// Mitsubishi GX Works2 project: Embotido   PLC: FX1S

// global labels: Global1
VAR_GLOBAL
  Sensor1 AT X002 : BOOL;
  Sensor2 AT X003 : BOOL;
  Sensor3 AT X005 : BOOL;
  Sensor4 AT X004 : BOOL;
  btnStart AT X000 : BOOL;
  btnStop AT X001 : BOOL;
  btnManConveyor AT X012 : BOOL;
  btnManSolenoid2 AT X007 : BOOL;
  btnManSolenoid1 AT X006 : BOOL;
  btnManSolenoid3 AT X010 : BOOL;
  btnManSolenoid4 AT X011 : BOOL;
  LightSensor1O AT Y007 : BOOL;
  LightSensor2O AT Y010 : BOOL;
  LightSensor3O AT Y011 : BOOL;
  LightSensor4O AT Y012 : BOOL;
  LightStartO AT Y005 : BOOL;
  LightStopO AT Y006 : BOOL;
  rConveyor AT Y004 : BOOL;
  rSolenoid1 AT Y000 : BOOL;
  rSolenoid2 AT Y001 : BOOL;
  rSolenoid4 AT Y003 : BOOL;
  rSolenoid3 AT Y002 : BOOL;
  runAutoFlag : BOOL;
  runAutoStatus : INT;
  conveyorRunFlag : BOOL;
  solenoid2RunFlag : BOOL;
  solenoid1RunFlag : BOOL;
  solenoid3RunFlag : BOOL;
  solenoid4RunFlag : BOOL;
  conveyorManRunFlag : BOOL;
  solenoid1ManRunFlag : BOOL;
  solenoid2ManRunFlag : BOOL;
  solenoid3ManRunFlag : BOOL;
  solenoid4ManRunFlag : BOOL;
END_VAR

// task Task_01 (event TRUE, interval 0, priority 31): POU_01

PROGRAM POU_01
VAR
  ConveyorRun : RunStop;
  Solenoid1Run : RunStop;
  Solenoid2Run : RunStop;
  Solenoid3Run : RunStop;
  Solenoid4Run : RunStop;
  ConveyorManualRun : StartStop;
  Solenoid1ManualRun : StartStop;
  Solenoid2ManualRun : StartStop;
  Solenoid3ManualRun : StartStop;
  Solenoid4ManualRun : StartStop;
  LightSensor1 : RunStop;
  LightSensor2 : RunStop;
  LightSensor3 : RunStop;
  LightSensor4 : RunStop;
  LightStart : RunStop;
  LightStop : RunStop;
END_VAR
(* START AUTO*)
IF btnStart = TRUE THEN
	runAutoFlag := TRUE;
	runAutoStatus := 1;
END_IF;
(* STOP AUTO*)
IF btnStop = TRUE THEN
	runAutoStatus := 0;

	runAutoFlag := FALSE;
	conveyorRunFlag := FALSE;
	solenoid1RunFlag := FALSE;
	solenoid2RunFlag := FALSE;
	solenoid3RunFlag := FALSE;
	solenoid4RunFlag := FALSE;
	conveyorManRunFlag := FALSE;
	solenoid1ManRunFlag := FALSE;
	solenoid2ManRunFlag := FALSE;
	solenoid3ManRunFlag := FALSE;
	solenoid4ManRunFlag := FALSE;
END_IF;

IF runAutoFlag = TRUE THEN
	conveyorManRunFlag = TRUE;
	
	IF Sensor1 = FALSE THEN
		solenoid1RunFlag := TRUE;
	ELSE
		solenoid1RunFlag := FALSE;
	END_IF;
	
	IF Sensor2 = FALSE THEN
		solenoid2RunFlag := TRUE;
	ELSE
		solenoid2RunFlag := FALSE;
	END_IF;
	
	IF Sensor3 = FALSE THEN
		solenoid3RunFlag := TRUE;
	ELSE
		solenoid3RunFlag := FALSE;
	END_IF;
	
	IF Sensor4 = FALSE THEN
		solenoid4RunFlag := TRUE;
	ELSE
		solenoid4RunFlag := FALSE;
	END_IF;
	
	ConveyorRun(input:= conveyorRunFlag,output:= rConveyor );
	Solenoid1Run(input:= solenoid1RunFlag,output:= rSolenoid1 );
	Solenoid2Run(input:= solenoid2RunFlag,output:= rSolenoid2 );
	Solenoid3Run(input:= solenoid3RunFlag,output:= rSolenoid3 );
	Solenoid4Run(input:= solenoid4RunFlag,output:= rSolenoid4 );
ELSE
	ConveyorManualRun(btnInput:= btnManConveyor ,memoryOn:= M1 ,memoryOff:= M2 ,memoryOutput:= conveyorManRunFlag );
	Solenoid1ManualRun(btnInput:= btnManSolenoid1 ,memoryOn:= M3 ,memoryOff:= M4 ,memoryOutput:= solenoid1ManRunFlag );
	Solenoid2ManualRun(btnInput:= btnManSolenoid2 ,memoryOn:= M5 ,memoryOff:= M6 ,memoryOutput:= solenoid2ManRunFlag  );
	Solenoid3ManualRun(btnInput:= btnManSolenoid3 ,memoryOn:= M7 ,memoryOff:= M8 ,memoryOutput:= solenoid3ManRunFlag  );
	Solenoid4ManualRun(btnInput:= btnManSolenoid4 ,memoryOn:= M9 ,memoryOff:= M10 ,memoryOutput:= solenoid4ManRunFlag  );
	
	ConveyorRun(input:= conveyorManRunFlag ,output:= rConveyor );
	Solenoid1Run(input:= solenoid1ManRunFlag ,output:= rSolenoid1 );
	Solenoid2Run(input:= solenoid2ManRunFlag ,output:= rSolenoid2 );
	Solenoid3Run(input:= solenoid3ManRunFlag ,output:= rSolenoid3 );
	Solenoid4Run(input:= solenoid4ManRunFlag ,output:= rSolenoid4 );
END_IF;

LightSensor1(input:= NOT Sensor1 ,output:=  LightSensor1O);
LightSensor2(input:= NOT Sensor2  ,output:= LightSensor2O );
LightSensor3(input:= NOT Sensor3  ,output:= LightSensor3O );
LightSensor4(input:= NOT Sensor4  ,output:= LightSensor4O );
LightStart(input:= runAutoFlag ,output:= LightStartO);
LightStop(input:= NOT runAutoFlag ,output:= LightStopO);
END_PROGRAM

FUNCTION_BLOCK StartStop
VAR_INPUT
  btnInput : BOOL;
END_VAR
VAR_IN_OUT
  memoryOn : BOOL;
  memoryOff : BOOL;
END_VAR
VAR_OUTPUT
  memoryOutput : BOOL;
END_VAR
(* structured ladder/FBD written out as ST: instructions are called as NAME(EN, inputs, outputs); _pN, _eN, _tN stand for wires *)
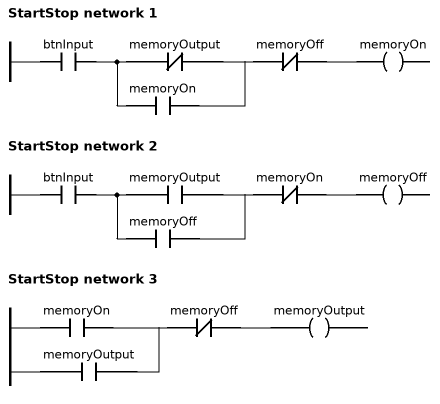
(* network 1 *)
memoryOn := ((btnInput AND NOT memoryOutput) OR (btnInput AND memoryOn)) AND NOT memoryOff;
(* network 2 *)
memoryOff := ((btnInput AND memoryOutput) OR (btnInput AND memoryOff)) AND NOT memoryOn;
(* network 3 *)
memoryOutput := (memoryOn OR memoryOutput) AND NOT memoryOff;
END_FUNCTION_BLOCK

FUNCTION_BLOCK RunStop
VAR_INPUT
  input : BOOL;
END_VAR
VAR_OUTPUT
  output : BOOL;
END_VAR
(* structured ladder/FBD written out as ST: instructions are called as NAME(EN, inputs, outputs); _pN, _eN, _tN stand for wires *)
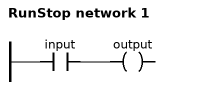
(* network 1 *)
output := input;
END_FUNCTION_BLOCK
